(*	Sample Code Disclaimer
	All sample code provided by Beckhoff Automation LLC are for illustrative purposes only
	and are provided “as is” and without any warranties, express or implied.
	Actual implementations in applications will vary significantly.
	Beckhoff Automation LLC shall have no liability for, and does not waive any rights in relation to,
	any code samples that it provides or the use of such code samples for any purpose.
*)
FUNCTION_BLOCK FB_StatFilter
VAR
	// Properties
	_Weight: UDINT := 1;
	_Count: UDINT;
	_Valid: BOOL;
	_LastValue: LREAL;
	_Minimum: LREAL;
	_Maximum: LREAL;
	_Avg: LREAL;
	_RMS: LREAL;
	_StdDev: LREAL;
	_StdErr: LREAL;
	
	rCount: LREAL;
	nIter: INT;
END_VAR

PROPERTY Avg : LREAL
GET
Avg := _Avg;
END_GET
END_PROPERTY

PROPERTY Count : UDINT
GET
Count := _Count;
END_GET
END_PROPERTY

PROPERTY LastValue : LREAL
GET
LastValue := _LastValue;
END_GET
END_PROPERTY

PROPERTY Maximum : LREAL
GET
Maximum := _Maximum;
END_GET
END_PROPERTY

PROPERTY Minimum : LREAL
GET
Minimum := _Minimum;
END_GET
END_PROPERTY

METHOD Reset : BOOL
VAR_INPUT
END_VAR

VAR
	
END_VAR
// Reset Stats
_Valid := FALSE;
_Count := 0;
_Minimum := 0;
_Maximum := 0;
_Avg := 0.0;
_StdDev := 0.0;
_StdErr := 0.0;
END_METHOD

PROPERTY RMS : LREAL
GET
RMS := _RMS;
END_GET
END_PROPERTY

METHOD Sample : BOOL
VAR_INPUT
	Value: lreal;
END_VAR
_Count := _Count +1;
IF _Count < _Weight OR _Weight = 0 THEN
	rCount := UDINT_TO_REAL(_Count);
ELSE
	_Valid := TRUE;
	rCount := UDINT_TO_REAL(_Weight);
END_IF

IF rCount > 0.0 THEN
	IF rCount = 1 OR Value < _Minimum THEN
		_Minimum := Value;
	END_IF
	
	IF rCount = 1 OR Value > _Maximum THEN
		_Maximum := Value;
	END_IF
	
	_Avg := (Value + _Avg * (rCount-1.0))/ rCount;
	_RMS := SQRT(  ( EXPT(Value,2)        + (rCount-1.0)*EXPT(_RMS,2)    ) / rCount  );
	_StdDev := SQRT(  ( EXPT(Value-_Avg,2) + (rCount-1.0)*EXPT(_StdDev,2) ) / rCount );
	_StdErr := _StdDev/ SQRT(rCount);

END_IF

_LastValue := Value;
END_METHOD

PROPERTY StdDev : LREAL
GET
StdDev := _StdDev;
END_GET
END_PROPERTY

PROPERTY StdErr : LREAL
GET
StdErr := _StdErr;
END_GET
END_PROPERTY

PROPERTY Valid : BOOL
GET
Valid := _Valid;
END_GET
END_PROPERTY

PROPERTY Weight : UDINT
GET
Weight := _Weight;
END_GET
SET
IF Weight <> _Weight THEN
	_Valid := FALSE;
	_Count := 0;
	_Minimum := 0;
	_Maximum := 0;
	_Avg := 0.0;
	_StdDev := 0.0;
	_StdErr := 0.0;
END_IF

_Weight := Weight;
END_SET
END_PROPERTY

END_FUNCTION_BLOCK

(* stored: Version 1.1.0.1, ProductVersion 3.1.4024.12
   POU FB_StatFilter: Id {4791098f-a430-4bbf-9d9f-5cbd2bc3f380}, SpecialFunc None
   Folder Stats: Id {6fbbf7dc-3719-4b86-ba7f-437abc40b4a5}
   Property Avg: Id {fb37e223-f2a4-4f05-9986-a7d28bcc5cc8}
   Get Get: Id {0b945e35-b92e-4905-ae00-e098ba6e961a}
   Property Count: Id {85298f51-76c4-48a0-aebf-2f4cfe248839}
   Get Get: Id {ee6a97ac-18bd-4a48-93d2-f9649805396e}
   Property LastValue: Id {018bd168-0c5b-42d4-a40f-29316ea66338}
   Get Get: Id {047b034b-a5f9-40d4-861b-9de89b617700}
   Property Maximum: Id {56a92ace-ecfa-4fa0-a6b7-b896b937cc16}
   Get Get: Id {94a7c02d-3da3-42a0-b9ba-c1df9efc541b}
   Property Minimum: Id {bab6c03d-18ac-4803-ad7a-12e2974edc21}
   Get Get: Id {1832b3ef-a367-4d0b-a055-852f21715bd1}
   Method Reset: Id {bf223b2b-781e-4bbe-b9bb-71ba57174884}
   Property RMS: Id {c8848003-4a0c-43ca-9dc0-2dab88c47fc5}
   Get Get: Id {6771b0ea-1568-4291-9a26-04694dc6bc62}
   Method Sample: Id {49850910-1ea1-442a-b5dd-8a3c132e652a}
   Property StdDev: Id {e074620f-958d-4b05-b7d5-b0e6e54f284f}
   Get Get: Id {0c7b7579-7558-4b84-aa7b-e449e6f1b293}
   Property StdErr: Id {a3e03c77-e759-4f05-adc9-7b8ce5ba4fd6}
   Get Get: Id {91f611f8-8ac5-41be-a8fc-84c4483cff11}
   Property Valid: Id {b6d3a36a-91f4-43dd-99d1-f489ba898092}
   Get Get: Id {3cb5d41e-d5fa-4074-9622-af1b5b30cf2f}
   Property Weight: Id {87e93b5d-c7b3-4969-87e7-f4e4e959fe2c}
   Get Get: Id {ebf50421-f94d-42b1-a91f-c7159b85490f}
   Set Set: Id {90d08384-4c78-4436-a070-134e6e7bcf64} *)
